INTERFACE I_Base1

METHOD metodo_base1 : BOOL
VAR_INPUT
END_VAR
END_METHOD

PROPERTY Prop_base1 : bool
GET
END_GET
SET
END_SET
END_PROPERTY

END_INTERFACE

(* stored: Version 1.1.0.1, ProductVersion 3.1.4024.12
   Itf I_Base1: Id {d7d1a935-1276-4e86-961b-270858c8a22a}
   Method metodo_base1: Id {58b92868-6280-40c8-a31a-2f7df4fe5190}
   Property Prop_base1: Id {7a786867-0cb6-48b1-86d6-1a9fdaa7428f}
   Get Get: Id {f6eebce0-4f41-4b9b-956a-5b30b5317f6e}
   Set Set: Id {c704e536-551b-4a23-a9f8-558e5c4ce018} *)
